// TIA Portal V17 export
// export: Created 2023-02-13T11:05:51.9872305Z, ExportSetting WithDefaults, DisplayName Totally Integrated Automation Portal, DisplayVersion V17, DisplayName TIA Portal Openness, DisplayVersion V17, DisplayName TIA Portal Teamcenter Gateway, DisplayVersion V17, DisplayName TIA Portal Version Control Interface, DisplayVersion V17, DisplayName SINAMICS Startdrive Advanced, DisplayVersion V17, DisplayName SINAMICS Startdrive G130, G150, S120, S150, SINAMICS MV, S210, DisplayVersion V17, DisplayName SINAMICS Startdrive G110M, G120, G120C, G120D, G120P, G115D, DisplayVersion V17, DisplayName STEP 7 Professional, DisplayVersion V17, DisplayName STEP 7 Safety, DisplayVersion V17, DisplayName WinCC Professional, DisplayVersion V17
VAR_GLOBAL   // PLC tag table "Default tag table"
   Tag_5 AT %QW746 : Word;
   Tag_6 AT %QW4750 : Word;
   System_Byte AT %MB1 : Byte;
   FirstScan AT %M1.0 : Bool;
   DiagStatusUpdate AT %M1.1 : Bool;
   AlwaysTRUE AT %M1.2 : Bool;
   AlwaysFALSE AT %M1.3 : Bool;
   Clock_Byte AT %MB0 : Byte;
   Clock_10Hz AT %M0.0 : Bool;
   Clock_5Hz AT %M0.1 : Bool;
   "Clock_2.5Hz" AT %M0.2 : Bool;
   Clock_2Hz AT %M0.3 : Bool;
   "Clock_1.25Hz" AT %M0.4 : Bool;
   Clock_1Hz AT %M0.5 : Bool;
   "Clock_0.625Hz" AT %M0.6 : Bool;
   "Clock_0.5Hz" AT %M0.7 : Bool;
   CryovacPotentioSP AT %MD1000 : Real;
   "FT-12.02_DUMMY" AT %MD1004 : Real;
   Tag_1 AT %M22.0 : Bool;
   ft1201pro AT %MD2000 : Real;
   Tag_2 AT %M1000.0 : Bool;
   Tag_3 AT %M1001.0 : Bool;
   ft1201hot AT %MD2006 : Real;
   Tag_4 AT %M3000.0 : Bool;
   "test BT Req" AT %M10.0 : Bool;
   TestLineTHE AT %M10.1 : Bool;
   "Timer 5S/1M" AT %M4.0 : Bool;
   "Timer 5S/30s" AT %M4.1 : Bool;
   Testing_FB_Valve_Prep AT %M100.0 : Bool;
   Tag_8 AT %M374.3 : Bool;
   Tag_9 AT %M999.0 : Bool;
   Tag_10 AT %MW990 : Word;
   Tag_11 AT %M400.0 : Bool;
   Tag_12 AT %M400.1 : Bool;
   Tag_13 AT %M400.2 : Bool;
   THE1_CommLBTimer AT %T1 : Timer;
   THE2_CommLBTimer AT %T2 : Timer;
   THE1_CommLBTimer1 AT %T3 : Timer;
   THE2_CommLBTimer1 AT %T4 : Timer;
   "Timer ON 5S" AT %T30 : Timer;
   "Timer OFF 1M" AT %T31 : Timer;
   "Timer ON 5S/30S" AT %T32 : Timer;
   "Timer OFF 30S" AT %T33 : Timer;
   timerDrainT61_MS AT %MD50 : Time;
   Testing_FB_Valve_Homo AT %M100.1 : Bool;
   Tag_7 AT %M100.2 : Bool;
   "Testing motor Prep" AT %M100.3 : Bool;
   Tag_14 AT %MD966 : Real;
   "Timer ON 10s/10s" AT %T5 : Timer;
   "Timer 8s/8s" AT %M4.2 : Bool;
   "Timer OFF 10s" AT %T6 : Timer;
   Tag_15 AT %M4.3 : Bool;
   Tag_16 AT %M4.4 : Bool;
   "CountMode_FT-12.01" AT %M5.0 : Bool;
   "CountMode_FT-12.02" AT %M5.1 : Bool;
   CountMode_HW_Blend AT %M5.3 : Bool;
   CountMode_ProWater_Blend AT %M5.2 : Bool;
   Tag_18 AT %M6.0 : Bool;
   Tag_19 AT %M7.0 : Bool;
END_VAR
